FUNCTION_BLOCK FB_Test_FSM EXTENDS TcUnit.FB_TestSuite
VAR_INPUT
END_VAR
VAR_OUTPUT
END_VAR
VAR
END_VAR

END_FUNCTION_BLOCK

(* stored: Version 1.1.0.1
   POU FB_Test_FSM: Id {eca0fa74-05f4-43bc-bf21-8752642e406c}, SpecialFunc None *)
